SUBAPPLICATION Ventilsteuerung_Uebung_010 (* SoftKey_F1 auf DigitalOutput_Q1 *)
  (* Standard: 61499-2 *)
  (* Version 1.0, 2023-10-23, franz *)
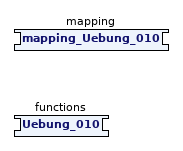
  SUBAPPS
    mapping : mapping_Uebung_010;
    functions : Uebung_010;
  END_SUBAPPS
END_SUBAPPLICATION
